# EPICS autosave request: sMailApp/Db/streamMail_settings.req
$(P)$(SM):addrTo
$(P)$(SM):addrFrom
